Fanuc KAREL source: kt00306.KL

-- PROVISIONAL review KL for V1013-1; original PC SHA256 11e45ab42e379a500236cf6e03f99f92a5c2aaa74d53c7ea351cecc108e65d3a
-- Incomplete behavior may be omitted. Consult companion uncertainty JSON. Do not deploy.
PROGRAM KT00306
%NOLOCKGROUP
VAR
  OUT : BOOLEAN
-- UNRESOLVED_DECL Y1 type=002018
-- UNRESOLVED_DECL H2 type=002017
BEGIN
  -- UNRESOLVED_PC offsets 5-19; opcodes 2E,22,9D,33,B2
  -- UNRESOLVED_PC offsets 24-38; opcodes 2E,22,9D,33,B4
  -- UNRESOLVED_PC offsets 43-68; opcodes 22,9D,33,B1,22,9D,33,B3,58,23
  -- UNRESOLVED_PC offsets 73-77; opcodes 7F
END KT00306
